FUNCTION_BLOCK OpenWebPage (* Composite Function Block Type *)
  (* Standard: 61499-2 *)
  (* Version 0.0, 6/26/2024, SESA685388, Schneider Electric, template *)
  PACKAGE SE.Nereda;
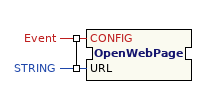
  EVENT_INPUT
    CONFIG WITH URL; (* Normal Execution Request *)
  END_EVENT
  VAR_INPUT
    URL : STRING := 'http://192.168.5.1'; (* Input event qualifier *)
  END_VAR
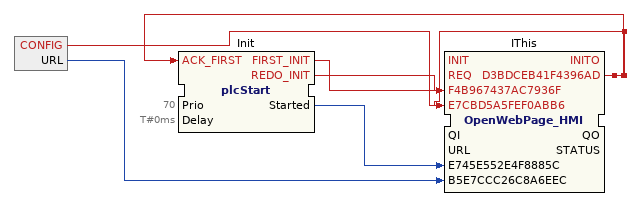
  (* 01 - FUNCTIONNAL INPUT INTERFACE *)
  (* 00 - INITIALIZATION *)
  (* 02 - FUNCTIONNAL OUTPUT INTERFACE *)
  (* 05 - LOGIC *)
  (* 06 - HMI INTERFACE *)
  (* 04 - CHILDREN *)
  (* 4A - TYPICALS *)
  (* 4B - SUBSYSTEMS *)
  (* 03 - FIELD INTERFACE *)
  (* 06 - IT/OT CONVERGENCE *)
  FBS
    Init : plcStart(Prio := 70, Delay := T#0ms);
    IThis : OpenWebPage_HMI;
  END_FBS
  EVENT_CONNECTIONS
    Init.FIRST_INIT TO IThis.F4B967437AC7936F;
    Init.REDO_INIT TO IThis.F4B967437AC7936F;
    CONFIG TO IThis.E7CBD5A5FEF0ABB6;
    IThis.D3BDCEB41F4396AD TO Init.ACK_FIRST;
    IThis.D3BDCEB41F4396AD TO IThis.E7CBD5A5FEF0ABB6;
  END_CONNECTIONS
  DATA_CONNECTIONS
    Init.Started TO IThis.E745E552E4F8885C;
    URL TO IThis.B5E7CCC26C8A6EEC;
  END_CONNECTIONS
END_FUNCTION_BLOCK
